// TIA Portal V19 export
VAR_GLOBAL   // PLC tag table "CVLV"
END_VAR
